// TIA Portal V19 export
TYPE "typeUnEmnPara"
// stored: Access Published
   STRUCT
      cm1Vfd206 : "typeVfdInterface";
      cm5AxisControl { S7_SetPoint := 'True'} : "typeAxisControlInterface";
   END_STRUCT;
END_TYPE
